PROGRAM MAIN
VAR
	test : BOOL;
END_VAR

test := NOT test;

END_PROGRAM

(* stored: Version 1.1.0.1
   POU MAIN: Id {4072e265-598f-46e4-9b94-10743c967f2e}, SpecialFunc None *)
